% RSLogix 500 project LVD210603_BaseOnly.RSS, saved by version 12.00.00.00 %
PROJECT "LINL0619"    % processor: MicroLogix 1400 %

PROGRAM FILES
  LAD 2 "MAIN"  62 rungs  % Main Program Routine %
  LAD 4 "ENABLES"  16 rungs
  LAD 5 "FEED"  11 rungs  % normal %
  LAD 6 "SPEEDS"  11 rungs
  LAD 7 "HSC BOT"  5 rungs
  LAD 8 "HSC TOP"  5 rungs
  LAD 9 "1 MS STI"  22 rungs  % high speed %
  LAD 10 "SHIFT BOT"  5 rungs
  LAD 11 "SHIFT TOP"  6 rungs
  LAD 12 "BOTOPTIC"  3 rungs
  LAD 13 "BOTOPTMES"  7 rungs
  LAD 81 "I1"  21 rungs
  LAD 82 "I1 RESULT"  8 rungs
  LAD 83 "I1 PASS"  6 rungs
  LAD 84 "I1 FAIL"  4 rungs
  LAD 85 "I1 ACQ"  9 rungs
  LAD 86 "I1 TESTER"  5 rungs
  LAD 87 "I1 TRIG"  5 rungs
  LAD 88 "NO FIFO"  1 rungs
  LAD 89 "NO FIFO"  1 rungs
  LAD 90 "I1 DATA"  3 rungs
  LAD 91 "I1 FAULT"  9 rungs
  LAD 92 "I1 FIX1"  5 rungs
  LAD 93 "I1 FIX2"  3 rungs
  LAD 94 "I2"  1 rungs
  LAD 95 "I2 RESULT"  1 rungs
  LAD 96 "I2 PASS"  1 rungs
  LAD 97 "I2 FAIL"  1 rungs
  LAD 98 "I2 ACQ"  1 rungs
  LAD 99 "I2 TESTER"  1 rungs
  LAD 100 "I2 TRIG"  1 rungs
  LAD 101 "I2 FIFOSET"  1 rungs
  LAD 102 "I2 FIFOGET"  1 rungs
  LAD 103 "I2 DATA"  1 rungs
  LAD 104 "I2 FAULT"  1 rungs
  LAD 105 "I2 FIX1"  1 rungs
  LAD 106 "I2 FIX2"  1 rungs
  LAD 107 "I3"  1 rungs
  LAD 108 "I3 RESULT"  1 rungs
  LAD 109 "I3 PASS"  1 rungs
  LAD 110 "I3 FAIL"  1 rungs
  LAD 111 "I3 ACQ"  1 rungs
  LAD 112 "I3 TESTER"  1 rungs
  LAD 113 "I3 TRIG"  1 rungs
  LAD 114 "I3 FIFOSET"  1 rungs
  LAD 115 "I3 FIFOGET"  1 rungs
  LAD 116 "I3 DATA"  1 rungs
  LAD 117 "I3 FAULT"  1 rungs
  LAD 118 "I3 FIX1"  1 rungs
  LAD 119 "I3 FIX2"  1 rungs
  LAD 120 "I4"  1 rungs
  LAD 121 "I4 RESULT"  1 rungs
  LAD 122 "I4 PASS"  1 rungs
  LAD 123 "I4 FAIL"  1 rungs
  LAD 124 "I4 ACQ"  1 rungs
  LAD 125 "I4 TESTER"  1 rungs
  LAD 126 "I4 TRIG"  1 rungs
  LAD 127 "I4 FIFOSET"  1 rungs
  LAD 128 "I4 FIFOGET"  1 rungs
  LAD 129 "I4 DATA"  1 rungs
  LAD 130 "I4 FAULT"  1 rungs
  LAD 131 "I4 FIX1"  1 rungs
  LAD 132 "I4 FIX2"  1 rungs
  LAD 135 "XFER"  3 rungs
  LAD 137 "TOPOPTIC"  15 rungs
  LAD 138 "TOPOPVERT"  13 rungs
  LAD 139 "TOPOPREAL"  19 rungs
  LAD 140 "TOPOPTEST"  8 rungs
  LAD 141 "TOPOPRANGE"  6 rungs
  LAD 142 "TOPOPRANGE"  6 rungs
  LAD 143 "TOPOPOKAY"  6 rungs
  LAD 144 "TESTINJECT"  8 rungs
  LAD 148 "I5"  21 rungs
  LAD 149 "I5 RESULT"  7 rungs
  LAD 150 "I5 PASS"  6 rungs
  LAD 151 "I5 FAIL"  4 rungs
  LAD 152 "I5 ACQ"  9 rungs
  LAD 153 "I5 TESTER"  5 rungs
  LAD 154 "I5 TRIG"  5 rungs
  LAD 155 "I5 FIFOSET"  10 rungs
  LAD 156 "I5 FIFOGET"  8 rungs
  LAD 157 "I5 DATA"  3 rungs
  LAD 158 "I5 FAULT"  9 rungs
  LAD 159 "I5 FIX1"  5 rungs
  LAD 160 "I5 FIX2"  3 rungs
  LAD 161 "I6"  21 rungs
  LAD 162 "I6 RESULT"  7 rungs
  LAD 163 "I6 PASS"  5 rungs
  LAD 164 "I6 FAIL"  3 rungs
  LAD 165 "I6 ACQ"  8 rungs
  LAD 166 "I6 TESTER"  5 rungs
  LAD 167 "I6 TRIG"  5 rungs
  LAD 168 "I6 FIFOSET"  9 rungs
  LAD 169 "I6 FIFOGET"  8 rungs
  LAD 170 "I6 DATA"  3 rungs
  LAD 171 "I6 FAULT"  9 rungs
  LAD 172 "I6 FIX1"  5 rungs
  LAD 173 "I6 FIX2"  3 rungs
  LAD 174 "I7"  21 rungs
  LAD 175 "I7 RESULT"  7 rungs
  LAD 176 "I7 PASS"  6 rungs
  LAD 177 "I7 FAIL"  4 rungs
  LAD 178 "I7 ACQ"  9 rungs
  LAD 179 "I7 TESTER"  5 rungs
  LAD 180 "I7 TRIG"  5 rungs
  LAD 181 "I7 FIFOSET"  9 rungs
  LAD 182 "I7 FIFOGET"  8 rungs
  LAD 183 "I7 DATA"  3 rungs
  LAD 184 "I7 FAULT"  9 rungs
  LAD 185 "I7 FIX1"  5 rungs
  LAD 186 "I7 FIX2"  3 rungs
  LAD 187 "I8"  22 rungs
  LAD 188 "I8 RESULT"  7 rungs
  LAD 189 "I8 PASS"  6 rungs
  LAD 190 "I8 FAIL"  4 rungs
  LAD 191 "I8 ACQ"  9 rungs
  LAD 192 "I8 TESTER"  5 rungs
  LAD 193 "I8 TRIG"  5 rungs
  LAD 194 "I8 FIFOSET"  9 rungs
  LAD 195 "I8 FIFOGET"  8 rungs
  LAD 196 "I8 DATA"  3 rungs
  LAD 197 "I8 FAULT"  9 rungs
  LAD 198 "I8 FIX1"  5 rungs
  LAD 199 "I8 FIX2"  3 rungs
  LAD 200 "PASS BLOW"  15 rungs
  LAD 235 "TESTTRIGS"  7 rungs  % highspeed test triggers, not necessary %
  LAD 236 "TESTTRIG1"  4 rungs
  LAD 237 "TESTTRIG2"  4 rungs
  LAD 238 "TESTTRIG3"  4 rungs
  LAD 239 "TESTTRIG4"  4 rungs
  LAD 240 "TESTTRIG5"  4 rungs
  LAD 241 "TESTTRIG6"  4 rungs
  LAD 242 "TESTTRIG7"  4 rungs
  LAD 243 "TESTTRIG8"  4 rungs
  LAD 244 "PACKAGER"  31 rungs  % normal %
  LAD 245 "NO PACKAGE"  8 rungs
  LAD 246 "RATE1"  9 rungs
  LAD 247 "RATE2"  6 rungs
  LAD 248 "RESET RATE"  6 rungs
  LAD 249 "NP STOP"  8 rungs  % stop on no good %
  LAD 250 "SPEED BOT"  8 rungs  % high speed %
  LAD 251 "SPEED TOP"  8 rungs  % high speed %
  LAD 252 "P BOT"  7 rungs  % high speed %
  LAD 253 "P TOP"  7 rungs  % high speed %
  LAD 254 "TOTALCOUNT"  4 rungs
  LAD 255 "SAVED"  4 rungs

DATA FILES
  O0 OUTPUT  6 elements
  I1 INPUT  8 elements
  S2 STATUS  66 elements
  B3 BINARY  256 elements
  T4 TIMER  45 elements
  C5 COUNTER  1 elements
  R6 CONTROL  30 elements
  N7 INTEGER  200 elements
  F8 FLOAT  1 elements
  L13 LONG  256 elements
  L19 RATE DATA  50 elements
  L20 I7TIMEFIFO  50 elements
  L21 I7POSFIFO  50 elements
  L22 I8TIMEFIFO  50 elements
  L23 I8POSFIFO  50 elements
  L30 INS5TIME  50 elements
  L31 INS5POS  50 elements
  L32 INS6TIME  50 elements
  L33 INS6POS  50 elements
  B34 BOT NG  128 elements
  B35 TOP NG  128 elements
  B36 BOTGOOD  128 elements
  B37 TOPGOOD1  128 elements
  B38 EX1 TEST  128 elements
  B39 TOPGOOD2  128 elements
  B40 EX2 TEST  128 elements
  B99 REMOVED IO  5 elements
  B100 NEW HMI B  100 elements
  N101 NEW HMI N  256 elements
  L102 NEW HMI L  256 elements

LADDER 2 "MAIN"    % Main Program Routine %
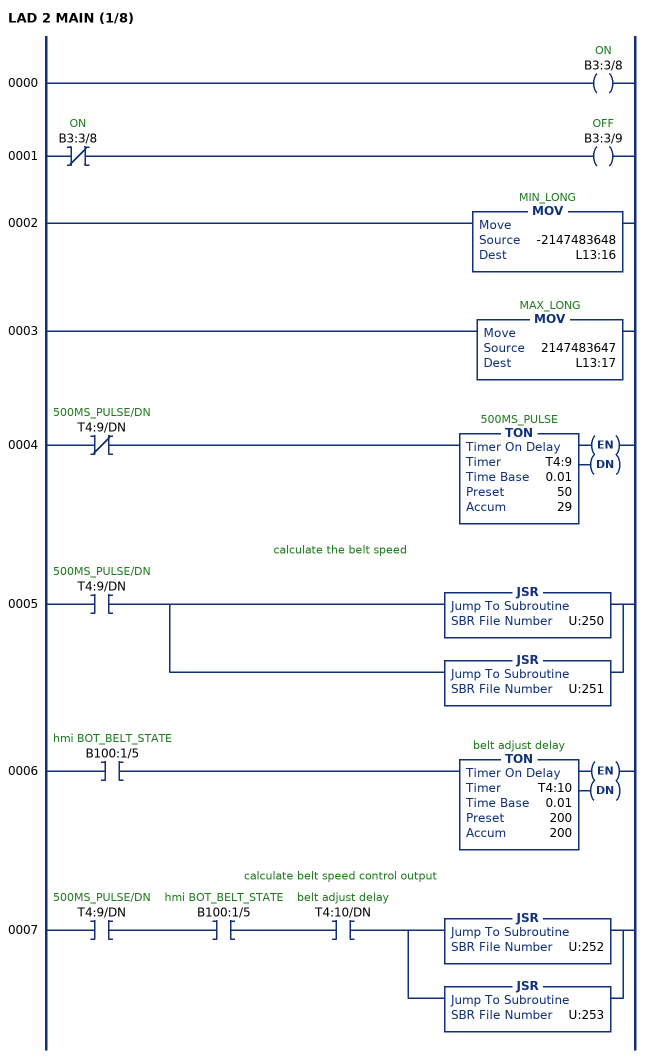
% Rung: 0 %
SOR OTE B3:3/8 EOR
%   B3:3/8  ON %
% Rung: 1 %
SOR XIO B3:3/8 OTE B3:3/9 EOR
%   B3:3/8  ON %
%   B3:3/9  OFF %
% Rung: 2 %
SOR MOV -2147483648 L13:16 EOR
%   L13:16  MIN_LONG %
% Rung: 3 %
SOR MOV 2147483647 L13:17 EOR
%   L13:17  MAX_LONG %
% Rung: 4 %
SOR XIO T4:9/DN TON T4:9 0.01 50 29 EOR
%   T4:9  500MS_PULSE %
% Rung: 5 %
% calculate the belt speed %
SOR XIC T4:9/DN BST JSR U:250 NXB JSR U:251 BND EOR
%   T4:9  500MS_PULSE %
% Rung: 6 %
SOR XIC B100:1/5 TON T4:10 0.01 200 200 EOR
%   B100:1/5  BOT_BELT_STATE  "hmi" %
%   T4:10  "belt adjust delay" %
% Rung: 7 %
% calculate belt speed control output %
SOR XIC T4:9/DN XIC B100:1/5 XIC T4:10/DN BST JSR U:252 NXB JSR U:253 BND EOR
%   T4:9  500MS_PULSE %
%   B100:1/5  BOT_BELT_STATE  "hmi" %
%   T4:10  "belt adjust delay" %

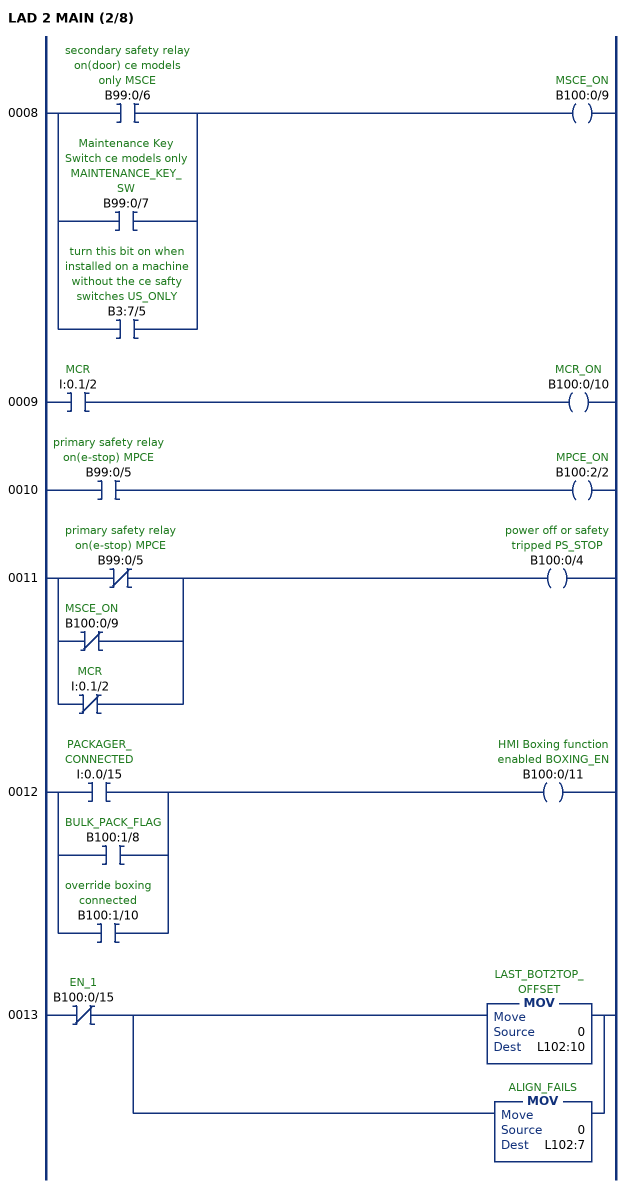
% Rung: 8 %
SOR BST XIC B99:0/6 NXB XIC B99:0/7 NXB XIC B3:7/5 BND OTE B100:0/9 EOR
%   B99:0/6  MSCE  "secondary safety relay on(door) ce models only" %
%   B99:0/7  MAINTENANCE_KEY_SW  "Maintenance Key Switch ce models only" %
%   B3:7/5  US_ONLY  "turn this bit on when installed on a machine without the ce safty switches" %
%   B100:0/9  MSCE_ON %
% Rung: 9 %
SOR XIC I:0.1/2 OTE B100:0/10 EOR
%   I:0.1/2  MCR %
%   B100:0/10  MCR_ON %
% Rung: 10 %
SOR XIC B99:0/5 OTE B100:2/2 EOR
%   B99:0/5  MPCE  "primary safety relay on(e-stop)" %
%   B100:2/2  MPCE_ON %
% Rung: 11 %
SOR BST XIO B99:0/5 NXB XIO B100:0/9 NXB XIO I:0.1/2 BND OTE B100:0/4 EOR
%   B99:0/5  MPCE  "primary safety relay on(e-stop)" %
%   B100:0/9  MSCE_ON %
%   I:0.1/2  MCR %
%   B100:0/4  PS_STOP  "power off or safety tripped" %
% Rung: 12 %
SOR BST XIC I:0.0/15 NXB XIC B100:1/8 NXB XIC B100:1/10 BND OTE B100:0/11 EOR
%   I:0.0/15  PACKAGER_CONNECTED %
%   B100:1/8  BULK_PACK_FLAG %
%   B100:1/10  "override boxing connected" %
%   B100:0/11  BOXING_EN  "HMI Boxing function enabled" %
% Rung: 13 %
SOR XIO B100:0/15 BST MOV 0 L102:10 NXB MOV 0 L102:7 BND EOR
%   B100:0/15  EN_1 %
%   L102:10  LAST_BOT2TOP_OFFSET %
%   L102:7  ALIGN_FAILS %

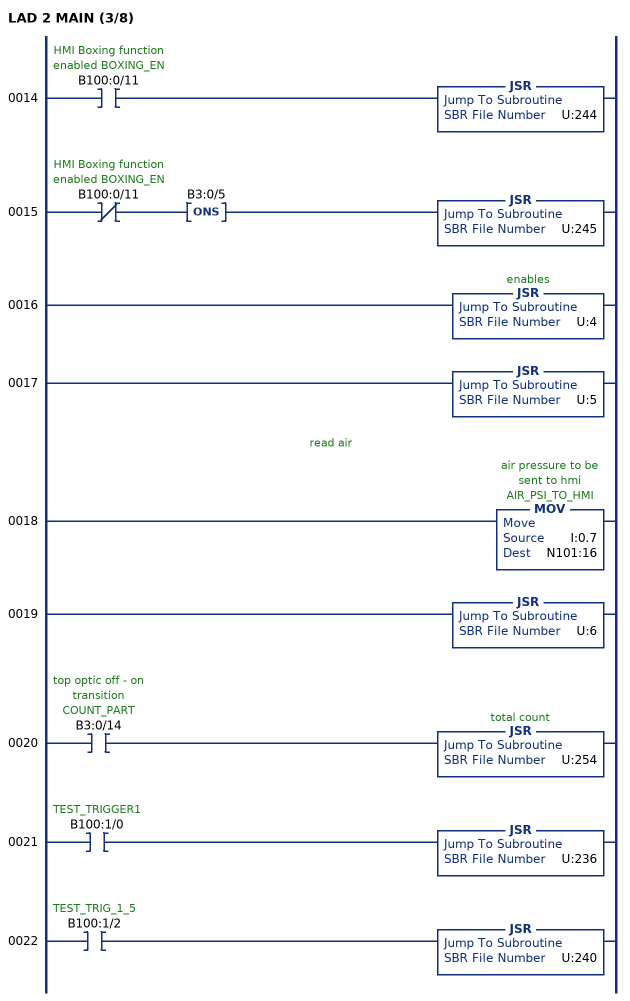
% Rung: 14 %
SOR XIC B100:0/11 JSR U:244 EOR
%   B100:0/11  BOXING_EN  "HMI Boxing function enabled" %
% Rung: 15 %
SOR XIO B100:0/11 ONS B3:0/5 JSR U:245 EOR
%   B100:0/11  BOXING_EN  "HMI Boxing function enabled" %
% Rung: 16 %
SOR JSR U:4 EOR
%   U:4  "enables" %
% Rung: 17 %
SOR JSR U:5 EOR
% Rung: 18 %
% read air %
SOR MOV I:0.7 N101:16 EOR
%   I:0.7  "Air Presure Sensor Input Signal" %
%   N101:16  AIR_PSI_TO_HMI  "air pressure to be sent to hmi" %
% Rung: 19 %
SOR JSR U:6 EOR
% Rung: 20 %
SOR XIC B3:0/14 JSR U:254 EOR
%   B3:0/14  COUNT_PART  "top optic off - on transition" %
%   U:254  "total count" %
% Rung: 21 %
SOR XIC B100:1/0 JSR U:236 EOR
%   B100:1/0  TEST_TRIGGER1 %
% Rung: 22 %
SOR XIC B100:1/2 JSR U:240 EOR
%   B100:1/2  TEST_TRIG_1_5 %

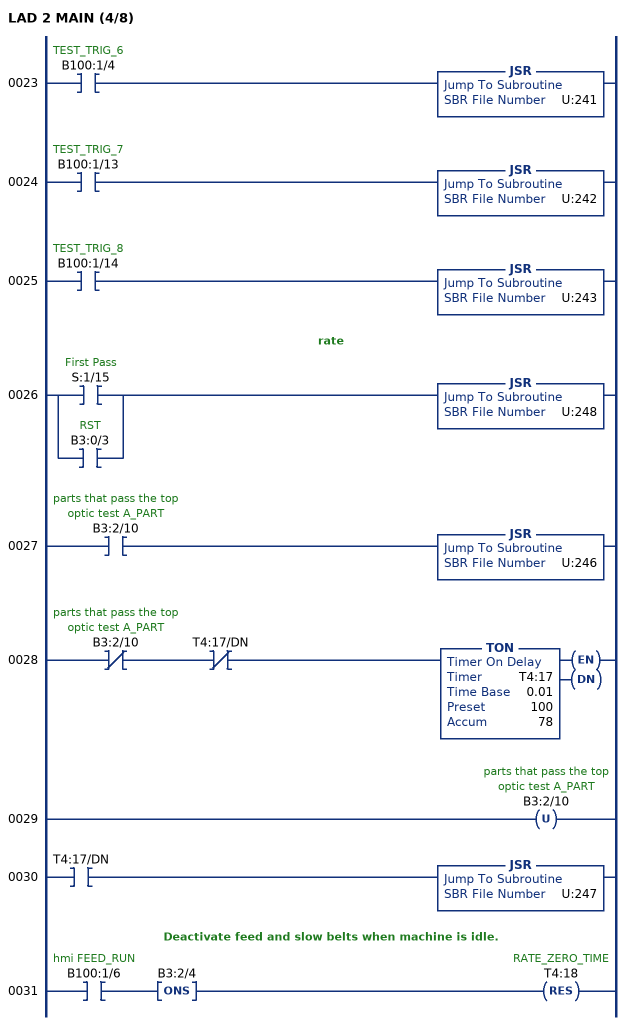
% Rung: 23 %
SOR XIC B100:1/4 JSR U:241 EOR
%   B100:1/4  TEST_TRIG_6 %
% Rung: 24 %
SOR XIC B100:1/13 JSR U:242 EOR
%   B100:1/13  TEST_TRIG_7 %
% Rung: 25 %
SOR XIC B100:1/14 JSR U:243 EOR
%   B100:1/14  TEST_TRIG_8 %
% Rung: 26 %
% TITLE: rate %
SOR BST XIC S:1/15 NXB XIC B3:0/3 BND JSR U:248 EOR
%   S:1/15  "First Pass" %
%   B3:0/3  RST %
% Rung: 27 %
SOR XIC B3:2/10 JSR U:246 EOR
%   B3:2/10  A_PART  "parts that pass the top optic test" %
% Rung: 28 %
SOR XIO B3:2/10 XIO T4:17/DN TON T4:17 0.01 100 78 EOR
%   B3:2/10  A_PART  "parts that pass the top optic test" %
% Rung: 29 %
SOR OTU B3:2/10 EOR
%   B3:2/10  A_PART  "parts that pass the top optic test" %
% Rung: 30 %
SOR XIC T4:17/DN JSR U:247 EOR
% Rung: 31 %
% TITLE: Deactivate feed and slow belts when machine is idle. %
SOR XIC B100:1/6 ONS B3:2/4 RES T4:18 EOR
%   B100:1/6  FEED_RUN  "hmi" %
%   T4:18  RATE_ZERO_TIME %

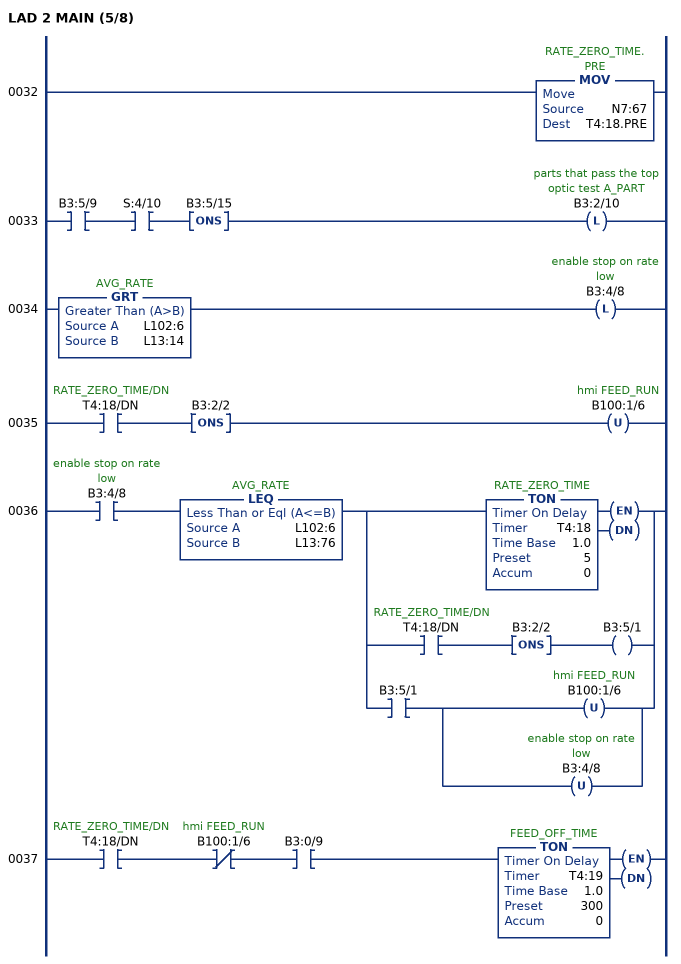
% Rung: 32 %
SOR MOV N7:67 T4:18.PRE EOR
%   N7:67  "empty bowl or jam bowl run time" %
%   T4:18  RATE_ZERO_TIME %
% Rung: 33 %
SOR XIC B3:5/9 XIC S:4/10 ONS B3:5/15 OTL B3:2/10 EOR
%   B3:2/10  A_PART  "parts that pass the top optic test" %
% Rung: 34 %
SOR GRT L102:6 L13:14 OTL B3:4/8 EOR
%   L102:6  AVG_RATE %
%   B3:4/8  "enable stop on rate low" %
% Rung: 35 %
SOR XIC T4:18/DN ONS B3:2/2 OTU B100:1/6 EOR
%   T4:18  RATE_ZERO_TIME %
%   B100:1/6  FEED_RUN  "hmi" %
% Rung: 36 %
SOR XIC B3:4/8 LEQ L102:6 L13:76 BST TON T4:18 1.0 5 0 NXB XIC T4:18/DN ONS B3:2/2 OTE B3:5/1 NXB XIC B3:5/1 BST OTU B100:1/6 NXB OTU B3:4/8 BND BND EOR
%   B3:4/8  "enable stop on rate low" %
%   L102:6  AVG_RATE %
%   T4:18  RATE_ZERO_TIME %
%   B100:1/6  FEED_RUN  "hmi" %
% Rung: 37 %
SOR XIC T4:18/DN XIO B100:1/6 XIC B3:0/9 TON T4:19 1.0 300 0 EOR
%   T4:18  RATE_ZERO_TIME %
%   B100:1/6  FEED_RUN  "hmi" %
%   T4:19  FEED_OFF_TIME %

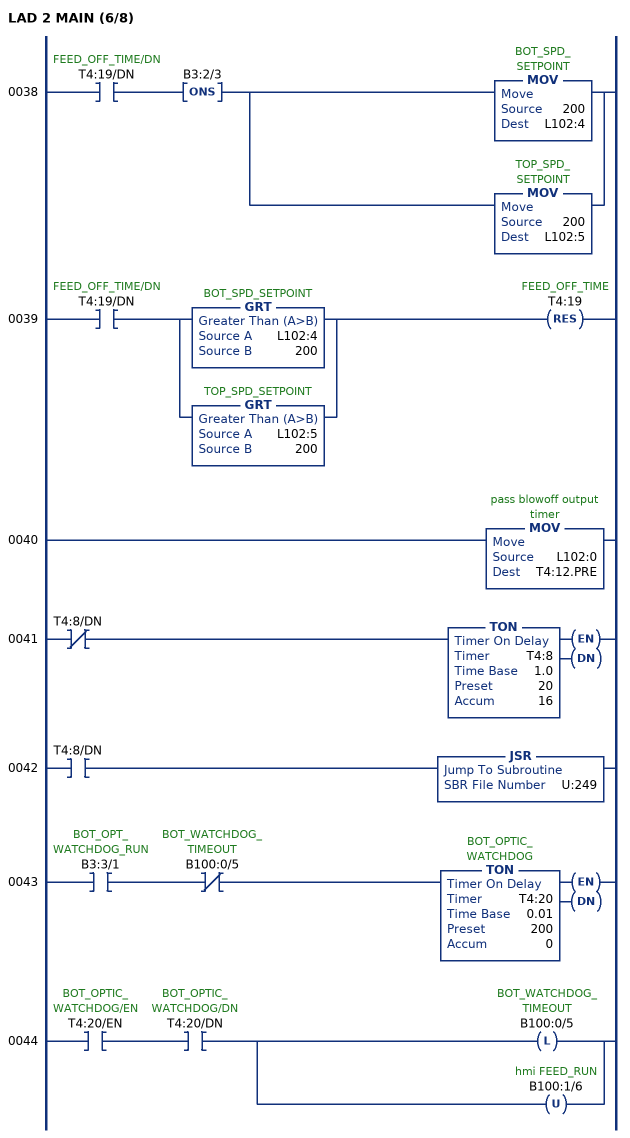
% Rung: 38 %
SOR XIC T4:19/DN ONS B3:2/3 BST MOV 200 L102:4 NXB MOV 200 L102:5 BND EOR
%   T4:19  FEED_OFF_TIME %
%   L102:4  BOT_SPD_SETPOINT %
%   L102:5  TOP_SPD_SETPOINT %
% Rung: 39 %
SOR XIC T4:19/DN BST GRT L102:4 200 NXB GRT L102:5 200 BND RES T4:19 EOR
%   T4:19  FEED_OFF_TIME %
%   L102:4  BOT_SPD_SETPOINT %
%   L102:5  TOP_SPD_SETPOINT %
% Rung: 40 %
SOR MOV L102:0 T4:12.PRE EOR
%   L102:0  BLOW_TIME %
%   T4:12  "pass blowoff output timer" %
% Rung: 41 %
SOR XIO T4:8/DN TON T4:8 1.0 20 16 EOR
% Rung: 42 %
SOR XIC T4:8/DN JSR U:249 EOR
% Rung: 43 %
SOR XIC B3:3/1 XIO B100:0/5 TON T4:20 0.01 200 0 EOR
%   B3:3/1  BOT_OPT_WATCHDOG_RUN %
%   B100:0/5  BOT_WATCHDOG_TIMEOUT %
%   T4:20  BOT_OPTIC_WATCHDOG %
% Rung: 44 %
SOR XIC T4:20/EN XIC T4:20/DN BST OTL B100:0/5 NXB OTU B100:1/6 BND EOR
%   T4:20  BOT_OPTIC_WATCHDOG %
%   B100:0/5  BOT_WATCHDOG_TIMEOUT %
%   B100:1/6  FEED_RUN  "hmi" %

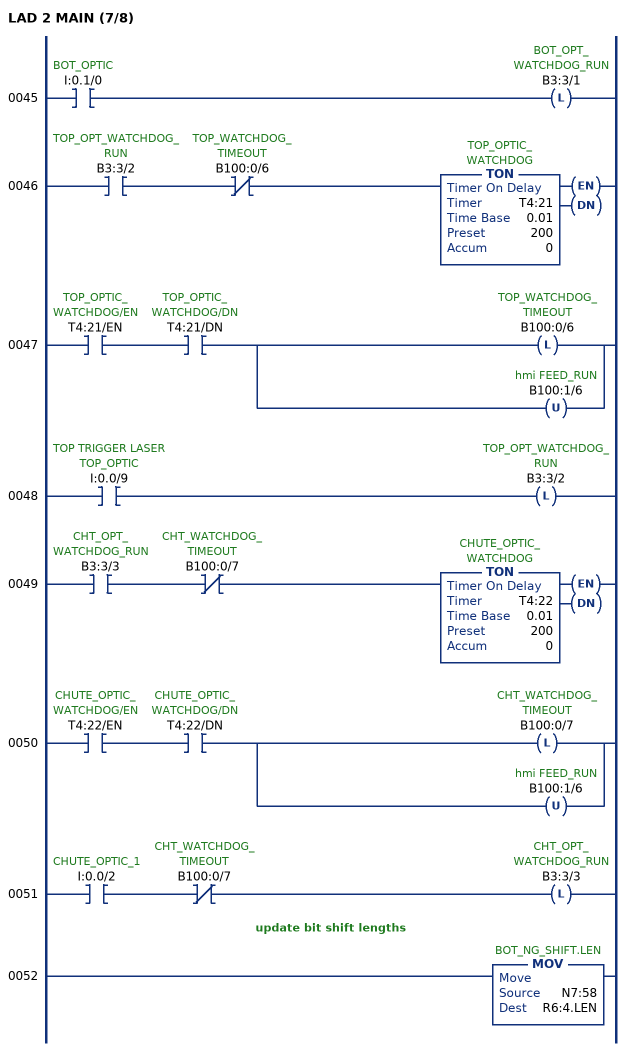
% Rung: 45 %
SOR XIC I:0.1/0 OTL B3:3/1 EOR
%   I:0.1/0  BOT_OPTIC %
%   B3:3/1  BOT_OPT_WATCHDOG_RUN %
% Rung: 46 %
SOR XIC B3:3/2 XIO B100:0/6 TON T4:21 0.01 200 0 EOR
%   B3:3/2  TOP_OPT_WATCHDOG_RUN %
%   B100:0/6  TOP_WATCHDOG_TIMEOUT %
%   T4:21  TOP_OPTIC_WATCHDOG %
% Rung: 47 %
SOR XIC T4:21/EN XIC T4:21/DN BST OTL B100:0/6 NXB OTU B100:1/6 BND EOR
%   T4:21  TOP_OPTIC_WATCHDOG %
%   B100:0/6  TOP_WATCHDOG_TIMEOUT %
%   B100:1/6  FEED_RUN  "hmi" %
% Rung: 48 %
SOR XIC I:0.0/9 OTL B3:3/2 EOR
%   I:0.0/9  TOP_OPTIC  "TOP TRIGGER LASER" %
%   B3:3/2  TOP_OPT_WATCHDOG_RUN %
% Rung: 49 %
SOR XIC B3:3/3 XIO B100:0/7 TON T4:22 0.01 200 0 EOR
%   B3:3/3  CHT_OPT_WATCHDOG_RUN %
%   B100:0/7  CHT_WATCHDOG_TIMEOUT %
%   T4:22  CHUTE_OPTIC_WATCHDOG %
% Rung: 50 %
SOR XIC T4:22/EN XIC T4:22/DN BST OTL B100:0/7 NXB OTU B100:1/6 BND EOR
%   T4:22  CHUTE_OPTIC_WATCHDOG %
%   B100:0/7  CHT_WATCHDOG_TIMEOUT %
%   B100:1/6  FEED_RUN  "hmi" %
% Rung: 51 %
SOR XIC I:0.0/2 XIO B100:0/7 OTL B3:3/3 EOR
%   I:0.0/2  CHUTE_OPTIC_1 %
%   B100:0/7  CHT_WATCHDOG_TIMEOUT %
%   B3:3/3  CHT_OPT_WATCHDOG_RUN %
% Rung: 52 %
% TITLE: update bit shift lengths %
SOR MOV N7:58 R6:4.LEN EOR
%   N7:58  BOT_NG_LENGTH %
%   R6:4  BOT_NG_SHIFT %

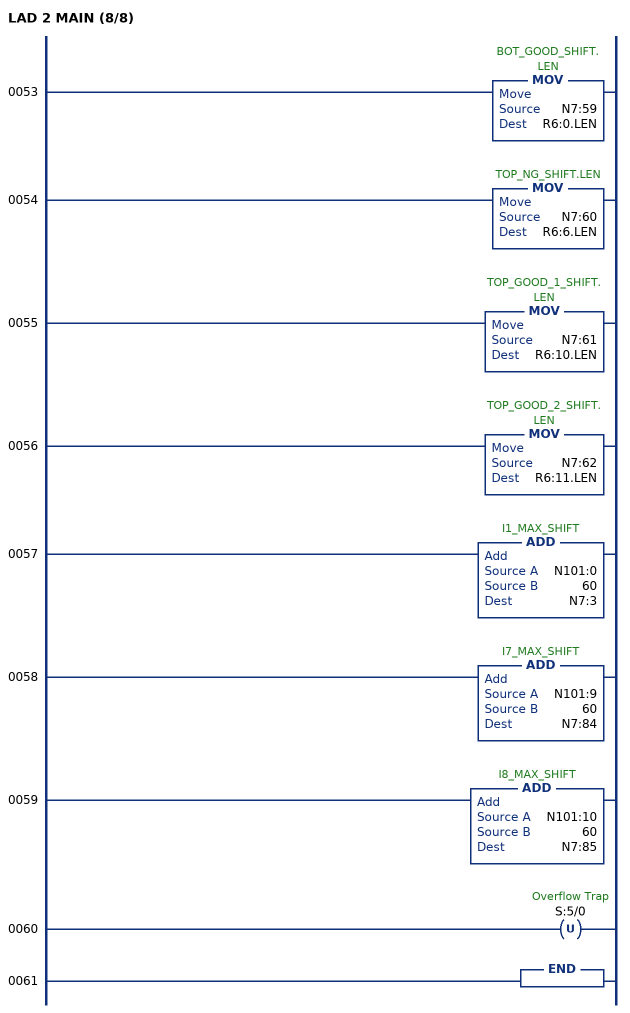
% Rung: 53 %
SOR MOV N7:59 R6:0.LEN EOR
%   N7:59  BOT_GOOD_LENGTH %
%   R6:0  BOT_GOOD_SHIFT %
% Rung: 54 %
SOR MOV N7:60 R6:6.LEN EOR
%   N7:60  TOP_NG_LENGTH %
%   R6:6  TOP_NG_SHIFT %
% Rung: 55 %
SOR MOV N7:61 R6:10.LEN EOR
%   N7:61  TOP_GOOD1_LENGTH %
%   R6:10  TOP_GOOD_1_SHIFT %
% Rung: 56 %
SOR MOV N7:62 R6:11.LEN EOR
%   N7:62  TOP_GOOD2_LENGTH %
%   R6:11  TOP_GOOD_2_SHIFT %
% Rung: 57 %
SOR ADD N101:0 60 N7:3 EOR
%   N101:0  I1_TRIG_LOC %
%   N7:3  I1_MAX_SHIFT %
% Rung: 58 %
SOR ADD N101:9 60 N7:84 EOR
%   N101:9  I7_TRIG_LOC %
%   N7:84  I7_MAX_SHIFT %
% Rung: 59 %
SOR ADD N101:10 60 N7:85 EOR
%   N101:10  I8_TRIG_LOC %
%   N7:85  I8_MAX_SHIFT %
% Rung: 60 %
SOR OTU S:5/0 EOR
%   S:5/0  "Overflow Trap" %
% Rung: 61 %
SOR END EOR

LADDER 4 "ENABLES"
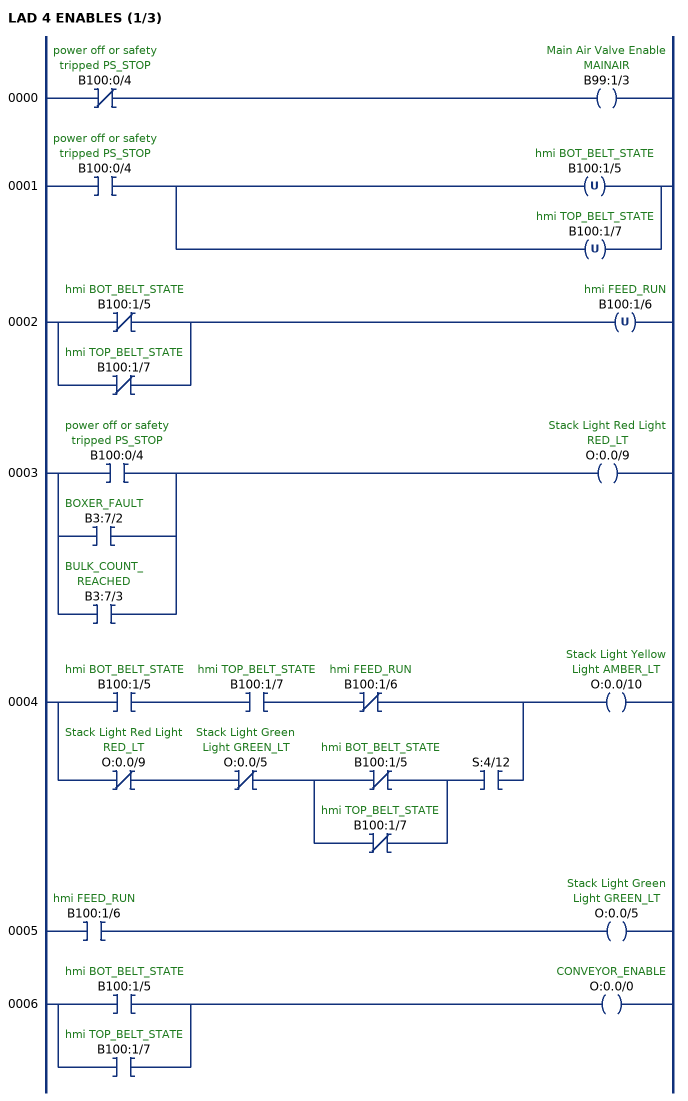
% Rung: 0 %
SOR XIO B100:0/4 OTE B99:1/3 EOR
%   B100:0/4  PS_STOP  "power off or safety tripped" %
%   B99:1/3  MAINAIR  "Main Air Valve Enable" %
% Rung: 1 %
SOR XIC B100:0/4 BST OTU B100:1/5 NXB OTU B100:1/7 BND EOR
%   B100:0/4  PS_STOP  "power off or safety tripped" %
%   B100:1/5  BOT_BELT_STATE  "hmi" %
%   B100:1/7  TOP_BELT_STATE  "hmi" %
% Rung: 2 %
SOR BST XIO B100:1/5 NXB XIO B100:1/7 BND OTU B100:1/6 EOR
%   B100:1/5  BOT_BELT_STATE  "hmi" %
%   B100:1/7  TOP_BELT_STATE  "hmi" %
%   B100:1/6  FEED_RUN  "hmi" %
% Rung: 3 %
SOR BST XIC B100:0/4 NXB XIC B3:7/2 NXB XIC B3:7/3 BND OTE O:0.0/9 EOR
%   B100:0/4  PS_STOP  "power off or safety tripped" %
%   B3:7/2  BOXER_FAULT %
%   B3:7/3  BULK_COUNT_REACHED %
%   O:0.0/9  RED_LT  "Stack Light Red Light" %
% Rung: 4 %
SOR BST XIC B100:1/5 XIC B100:1/7 XIO B100:1/6 NXB XIO O:0.0/9 XIO O:0.0/5 BST XIO B100:1/5 NXB XIO B100:1/7 BND XIC S:4/12 BND OTE O:0.0/10 EOR
%   B100:1/5  BOT_BELT_STATE  "hmi" %
%   B100:1/7  TOP_BELT_STATE  "hmi" %
%   B100:1/6  FEED_RUN  "hmi" %
%   O:0.0/9  RED_LT  "Stack Light Red Light" %
%   O:0.0/5  GREEN_LT  "Stack Light Green Light" %
%   O:0.0/10  AMBER_LT  "Stack Light Yellow Light" %
% Rung: 5 %
SOR XIC B100:1/6 OTE O:0.0/5 EOR
%   B100:1/6  FEED_RUN  "hmi" %
%   O:0.0/5  GREEN_LT  "Stack Light Green Light" %
% Rung: 6 %
SOR BST XIC B100:1/5 NXB XIC B100:1/7 BND OTE O:0.0/0 EOR
%   B100:1/5  BOT_BELT_STATE  "hmi" %
%   B100:1/7  TOP_BELT_STATE  "hmi" %
%   O:0.0/0  CONVEYOR_ENABLE %

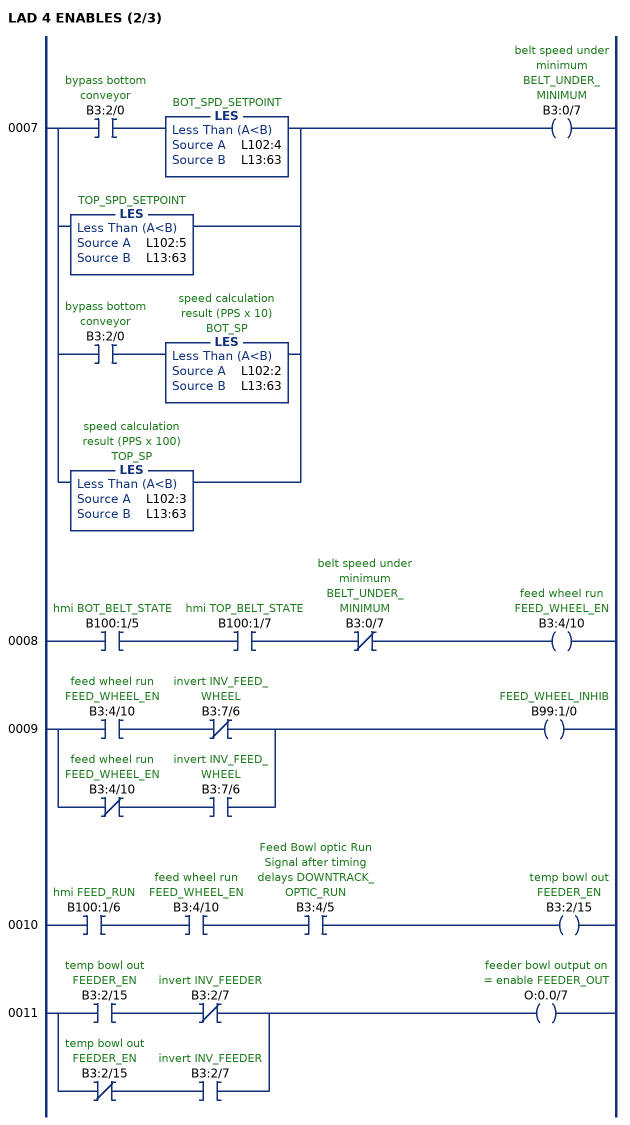
% Rung: 7 %
SOR BST XIC B3:2/0 LES L102:4 L13:63 NXB LES L102:5 L13:63 NXB XIC B3:2/0 LES L102:2 L13:63 NXB LES L102:3 L13:63 BND OTE B3:0/7 EOR
%   B3:2/0  "bypass bottom conveyor" %
%   L102:4  BOT_SPD_SETPOINT %
%   L13:63  "min belt speed" %
%   L102:5  TOP_SPD_SETPOINT %
%   L102:2  BOT_SP  "speed calculation result (PPS x 10)" %
%   L102:3  TOP_SP  "speed calculation result (PPS x 100)" %
%   B3:0/7  BELT_UNDER_MINIMUM  "belt speed under minimum" %
% Rung: 8 %
SOR XIC B100:1/5 XIC B100:1/7 XIO B3:0/7 OTE B3:4/10 EOR
%   B100:1/5  BOT_BELT_STATE  "hmi" %
%   B100:1/7  TOP_BELT_STATE  "hmi" %
%   B3:0/7  BELT_UNDER_MINIMUM  "belt speed under minimum" %
%   B3:4/10  FEED_WHEEL_EN  "feed wheel run" %
% Rung: 9 %
SOR BST XIC B3:4/10 XIO B3:7/6 NXB XIO B3:4/10 XIC B3:7/6 BND OTE B99:1/0 EOR
%   B3:4/10  FEED_WHEEL_EN  "feed wheel run" %
%   B3:7/6  INV_FEED_WHEEL  "invert" %
%   B99:1/0  FEED_WHEEL_INHIB %
% Rung: 10 %
SOR XIC B100:1/6 XIC B3:4/10 XIC B3:4/5 OTE B3:2/15 EOR
%   B100:1/6  FEED_RUN  "hmi" %
%   B3:4/10  FEED_WHEEL_EN  "feed wheel run" %
%   B3:4/5  DOWNTRACK_OPTIC_RUN  "Feed Bowl optic Run Signal after timing delays" %
%   B3:2/15  FEEDER_EN  "temp bowl out" %
% Rung: 11 %
SOR BST XIC B3:2/15 XIO B3:2/7 NXB XIO B3:2/15 XIC B3:2/7 BND OTE O:0.0/7 EOR
%   B3:2/15  FEEDER_EN  "temp bowl out" %
%   B3:2/7  INV_FEEDER  "invert" %
%   O:0.0/7  FEEDER_OUT  "feeder bowl output on = enable" %

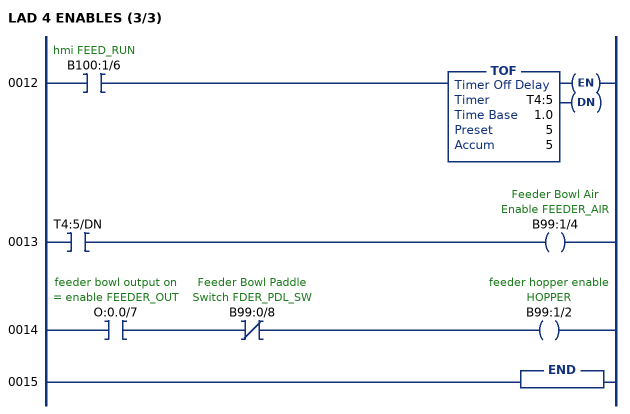
% Rung: 12 %
SOR XIC B100:1/6 TOF T4:5 1.0 5 5 EOR
%   B100:1/6  FEED_RUN  "hmi" %
% Rung: 13 %
SOR XIC T4:5/DN OTE B99:1/4 EOR
%   B99:1/4  FEEDER_AIR  "Feeder Bowl Air Enable" %
% Rung: 14 %
SOR XIC O:0.0/7 XIO B99:0/8 OTE B99:1/2 EOR
%   O:0.0/7  FEEDER_OUT  "feeder bowl output on = enable" %
%   B99:0/8  FDER_PDL_SW  "Feeder Bowl Paddle Switch" %
%   B99:1/2  HOPPER  "feeder hopper enable" %
% Rung: 15 %
SOR END EOR

LADDER 5 "FEED"    % normal %
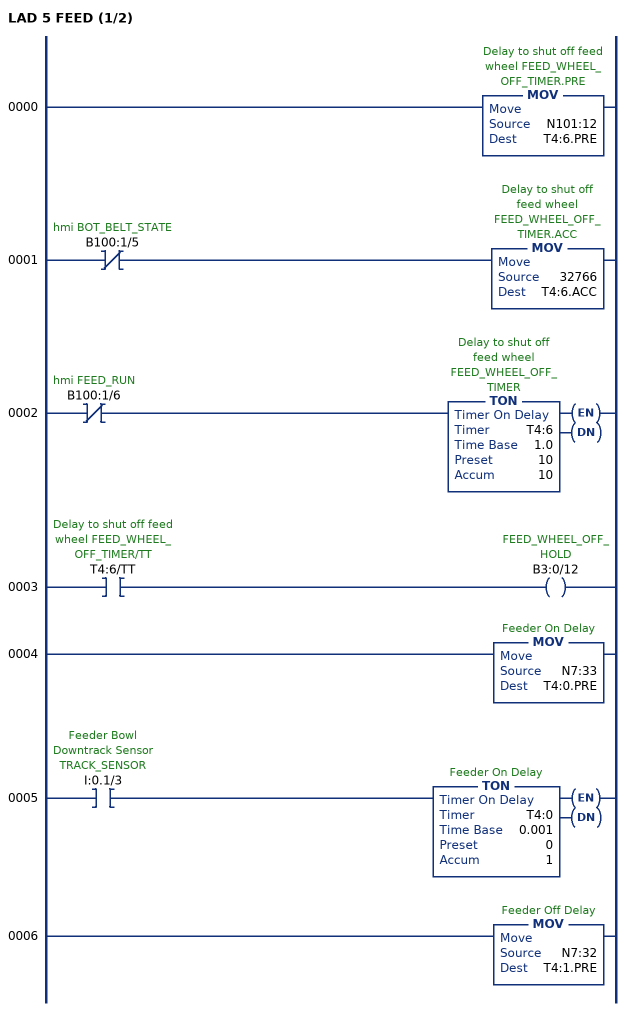
% Rung: 0 %
SOR MOV N101:12 T4:6.PRE EOR
%   N101:12  FEED_WHEEL_STOP_TIME %
%   T4:6  FEED_WHEEL_OFF_TIMER  "Delay to shut off feed wheel" %
% Rung: 1 %
SOR XIO B100:1/5 MOV 32766 T4:6.ACC EOR
%   B100:1/5  BOT_BELT_STATE  "hmi" %
%   T4:6  FEED_WHEEL_OFF_TIMER  "Delay to shut off feed wheel" %
% Rung: 2 %
SOR XIO B100:1/6 TON T4:6 1.0 10 10 EOR
%   B100:1/6  FEED_RUN  "hmi" %
%   T4:6  FEED_WHEEL_OFF_TIMER  "Delay to shut off feed wheel" %
% Rung: 3 %
SOR XIC T4:6/TT OTE B3:0/12 EOR
%   T4:6  FEED_WHEEL_OFF_TIMER  "Delay to shut off feed wheel" %
%   B3:0/12  FEED_WHEEL_OFF_HOLD %
% Rung: 4 %
SOR MOV N7:33 T4:0.PRE EOR
%   N7:33  "down track on delay" %
%   T4:0  "Feeder On Delay" %
% Rung: 5 %
SOR XIC I:0.1/3 TON T4:0 0.001 0 1 EOR
%   I:0.1/3  TRACK_SENSOR  "Feeder Bowl Downtrack Sensor" %
%   T4:0  "Feeder On Delay" %
% Rung: 6 %
SOR MOV N7:32 T4:1.PRE EOR
%   N7:32  "down track off delay" %
%   T4:1  "Feeder Off Delay" %

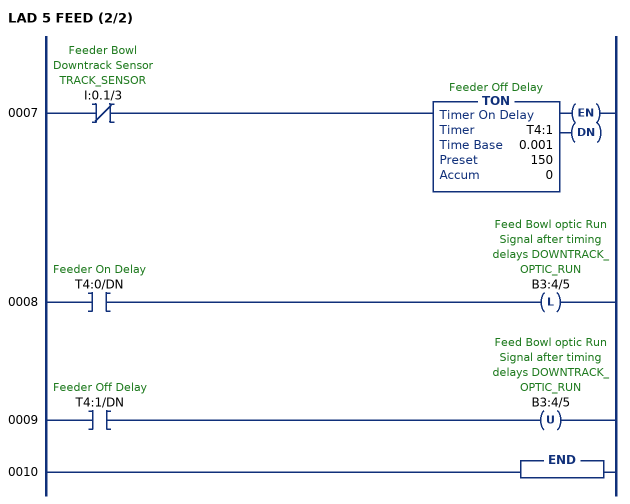
% Rung: 7 %
SOR XIO I:0.1/3 TON T4:1 0.001 150 0 EOR
%   I:0.1/3  TRACK_SENSOR  "Feeder Bowl Downtrack Sensor" %
%   T4:1  "Feeder Off Delay" %
% Rung: 8 %
SOR XIC T4:0/DN OTL B3:4/5 EOR
%   T4:0  "Feeder On Delay" %
%   B3:4/5  DOWNTRACK_OPTIC_RUN  "Feed Bowl optic Run Signal after timing delays" %
% Rung: 9 %
SOR XIC T4:1/DN OTU B3:4/5 EOR
%   T4:1  "Feeder Off Delay" %
%   B3:4/5  DOWNTRACK_OPTIC_RUN  "Feed Bowl optic Run Signal after timing delays" %
% Rung: 10 %
SOR END EOR

LADDER 6 "SPEEDS"
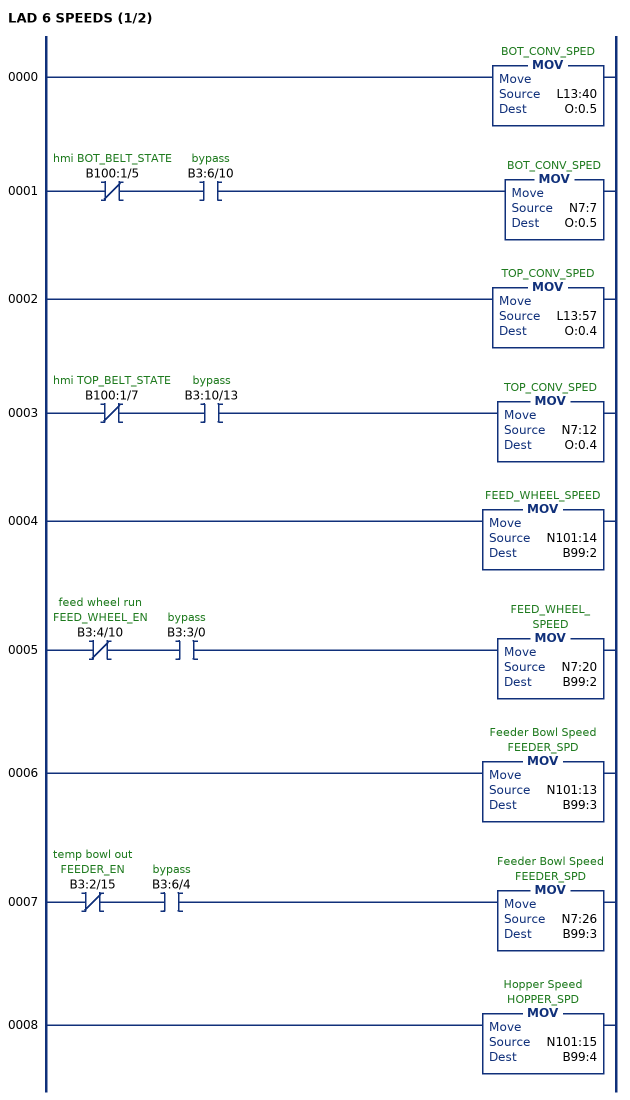
% Rung: 0 %
SOR MOV L13:40 O:0.5 EOR
%   L13:40  SCALED_BOT_VALUE %
%   O:0.5  BOT_CONV_SPED %
% Rung: 1 %
SOR XIO B100:1/5 XIC B3:6/10 MOV N7:7 O:0.5 EOR
%   B100:1/5  BOT_BELT_STATE  "hmi" %
%   B3:6/10  "bypass" %
%   O:0.5  BOT_CONV_SPED %
% Rung: 2 %
SOR MOV L13:57 O:0.4 EOR
%   L13:57  SCALED_TOP_VALUE %
%   O:0.4  TOP_CONV_SPED %
% Rung: 3 %
SOR XIO B100:1/7 XIC B3:10/13 MOV N7:12 O:0.4 EOR
%   B100:1/7  TOP_BELT_STATE  "hmi" %
%   B3:10/13  "bypass" %
%   O:0.4  TOP_CONV_SPED %
% Rung: 4 %
SOR MOV N101:14 B99:2 EOR
%   N101:14  FEED_WHL_SPD_SET  "feed wheel speed setting from hmi" %
%   B99:2  FEED_WHEEL_SPEED %
% Rung: 5 %
SOR XIO B3:4/10 XIC B3:3/0 MOV N7:20 B99:2 EOR
%   B3:4/10  FEED_WHEEL_EN  "feed wheel run" %
%   B3:3/0  "bypass" %
%   B99:2  FEED_WHEEL_SPEED %
% Rung: 6 %
SOR MOV N101:13 B99:3 EOR
%   N101:13  FEED_BOWL_SET_SPD %
%   B99:3  FEEDER_SPD  "Feeder Bowl Speed" %
% Rung: 7 %
SOR XIO B3:2/15 XIC B3:6/4 MOV N7:26 B99:3 EOR
%   B3:2/15  FEEDER_EN  "temp bowl out" %
%   B3:6/4  "bypass" %
%   B99:3  FEEDER_SPD  "Feeder Bowl Speed" %
% Rung: 8 %
SOR MOV N101:15 B99:4 EOR
%   N101:15  HOPPER_SPD_SET  "hopper speed setting from hmi" %
%   B99:4  HOPPER_SPD  "Hopper Speed" %

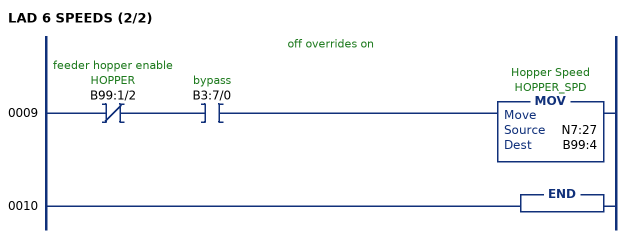
% Rung: 9 %
% off overrides on %
SOR XIO B99:1/2 XIC B3:7/0 MOV N7:27 B99:4 EOR
%   B99:1/2  HOPPER  "feeder hopper enable" %
%   B3:7/0  "bypass" %
%   B99:4  HOPPER_SPD  "Hopper Speed" %
% Rung: 10 %
SOR END EOR

LADDER 7 "HSC BOT"
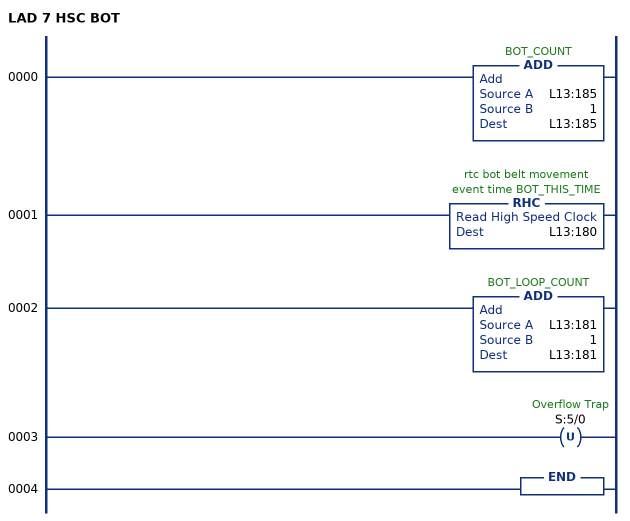
% Rung: 0 %
SOR ADD L13:185 1 L13:185 EOR
%   L13:185  BOT_COUNT %
% Rung: 1 %
SOR RHC L13:180 EOR
%   L13:180  BOT_THIS_TIME  "rtc bot belt movement event time" %
% Rung: 2 %
SOR ADD L13:181 1 L13:181 EOR
%   L13:181  BOT_LOOP_COUNT %
% Rung: 3 %
SOR OTU S:5/0 EOR
%   S:5/0  "Overflow Trap" %
% Rung: 4 %
SOR END EOR

LADDER 8 "HSC TOP"
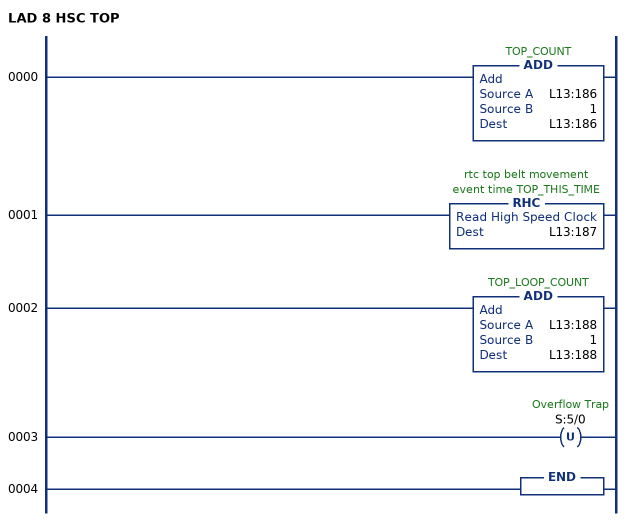
% Rung: 0 %
SOR ADD L13:186 1 L13:186 EOR
%   L13:186  TOP_COUNT %
% Rung: 1 %
SOR RHC L13:187 EOR
%   L13:187  TOP_THIS_TIME  "rtc top belt movement event time" %
% Rung: 2 %
SOR ADD L13:188 1 L13:188 EOR
%   L13:188  TOP_LOOP_COUNT %
% Rung: 3 %
SOR OTU S:5/0 EOR
%   S:5/0  "Overflow Trap" %
% Rung: 4 %
SOR END EOR

LADDER 9 "1 MS STI"    % high speed %
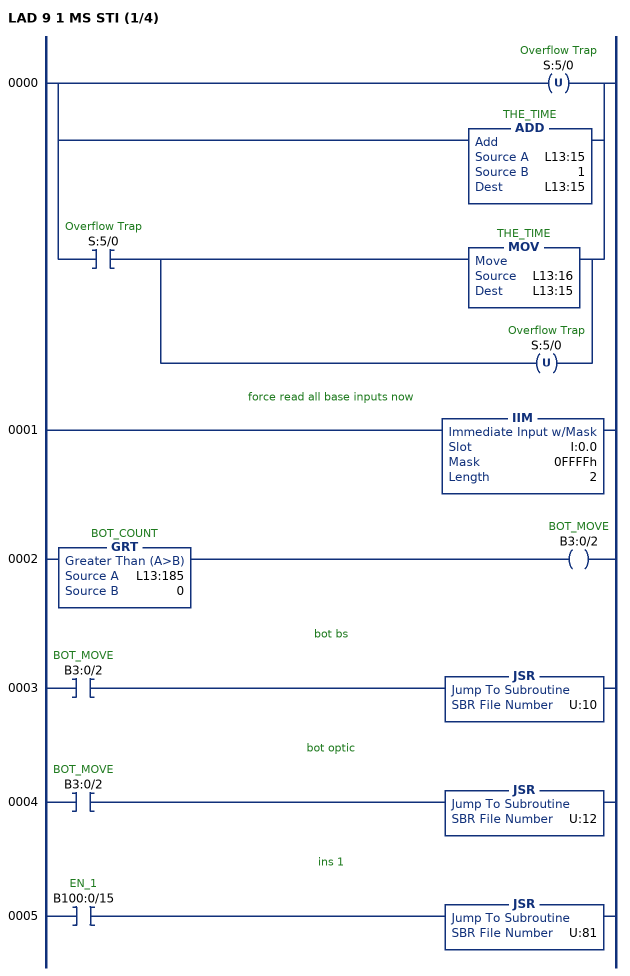
% Rung: 0 %
SOR BST OTU S:5/0 NXB ADD L13:15 1 L13:15 NXB XIC S:5/0 BST MOV L13:16 L13:15 NXB OTU S:5/0 BND BND EOR
%   S:5/0  "Overflow Trap" %
%   L13:15  THE_TIME %
%   L13:16  MIN_LONG %
% Rung: 1 %
% force read all base inputs now %
SOR IIM I:0.0 0FFFFh 2 EOR
% Rung: 2 %
SOR GRT L13:185 0 OTE B3:0/2 EOR
%   L13:185  BOT_COUNT %
%   B3:0/2  BOT_MOVE %
% Rung: 3 %
% bot bs %
SOR XIC B3:0/2 JSR U:10 EOR
%   B3:0/2  BOT_MOVE %
% Rung: 4 %
% bot optic %
SOR XIC B3:0/2 JSR U:12 EOR
%   B3:0/2  BOT_MOVE %
% Rung: 5 %
% ins 1 %
SOR XIC B100:0/15 JSR U:81 EOR
%   B100:0/15  EN_1 %

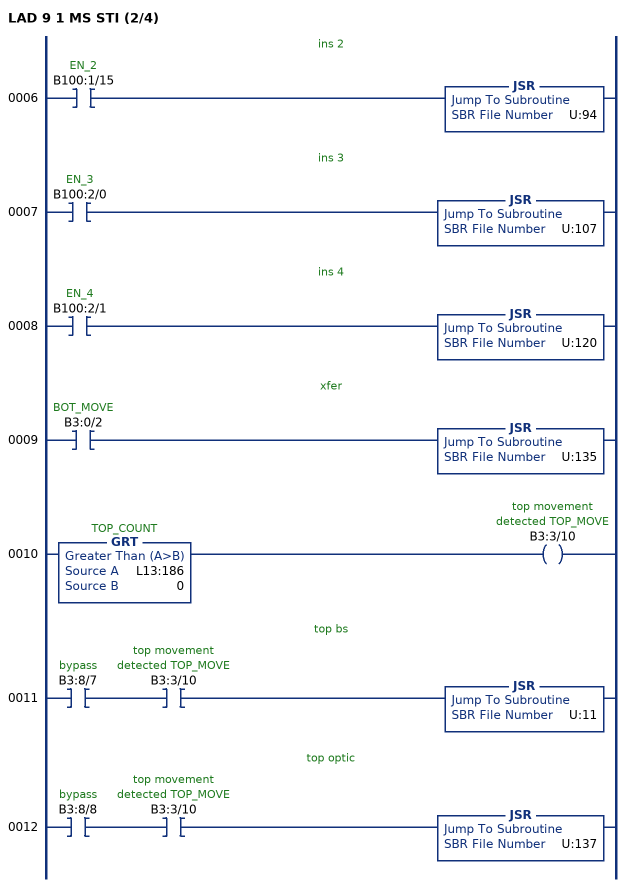
% Rung: 6 %
% ins 2 %
SOR XIC B100:1/15 JSR U:94 EOR
%   B100:1/15  EN_2 %
% Rung: 7 %
% ins 3 %
SOR XIC B100:2/0 JSR U:107 EOR
%   B100:2/0  EN_3 %
% Rung: 8 %
% ins 4 %
SOR XIC B100:2/1 JSR U:120 EOR
%   B100:2/1  EN_4 %
% Rung: 9 %
% xfer %
SOR XIC B3:0/2 JSR U:135 EOR
%   B3:0/2  BOT_MOVE %
% Rung: 10 %
SOR GRT L13:186 0 OTE B3:3/10 EOR
%   L13:186  TOP_COUNT %
%   B3:3/10  TOP_MOVE  "top movement detected" %
% Rung: 11 %
% top bs %
SOR XIC B3:8/7 XIC B3:3/10 JSR U:11 EOR
%   B3:8/7  "bypass" %
%   B3:3/10  TOP_MOVE  "top movement detected" %
% Rung: 12 %
% top optic %
SOR XIC B3:8/8 XIC B3:3/10 JSR U:137 EOR
%   B3:8/8  "bypass" %
%   B3:3/10  TOP_MOVE  "top movement detected" %

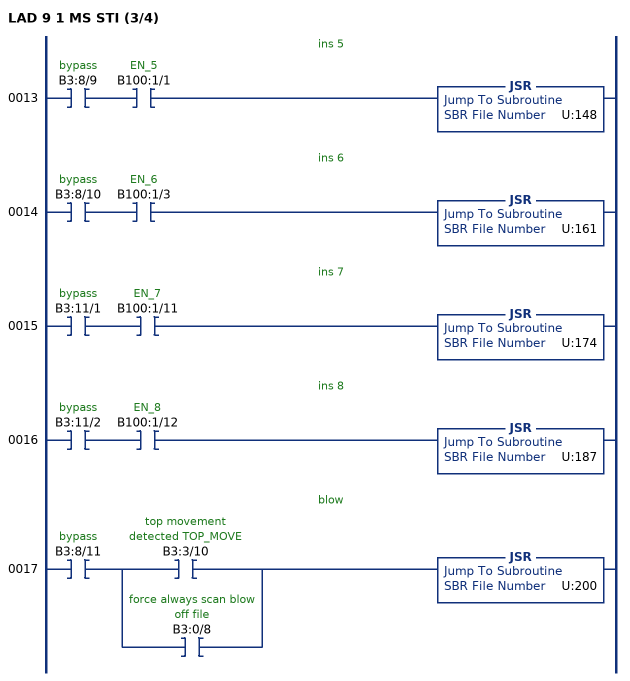
% Rung: 13 %
% ins 5 %
SOR XIC B3:8/9 XIC B100:1/1 JSR U:148 EOR
%   B3:8/9  "bypass" %
%   B100:1/1  EN_5 %
% Rung: 14 %
% ins 6 %
SOR XIC B3:8/10 XIC B100:1/3 JSR U:161 EOR
%   B3:8/10  "bypass" %
%   B100:1/3  EN_6 %
% Rung: 15 %
% ins 7 %
SOR XIC B3:11/1 XIC B100:1/11 JSR U:174 EOR
%   B3:11/1  "bypass" %
%   B100:1/11  EN_7 %
% Rung: 16 %
% ins 8 %
SOR XIC B3:11/2 XIC B100:1/12 JSR U:187 EOR
%   B3:11/2  "bypass" %
%   B100:1/12  EN_8 %
% Rung: 17 %
% blow %
SOR XIC B3:8/11 BST XIC B3:3/10 NXB XIC B3:0/8 BND JSR U:200 EOR
%   B3:8/11  "bypass" %
%   B3:3/10  TOP_MOVE  "top movement detected" %
%   B3:0/8  "force always scan blow off file" %

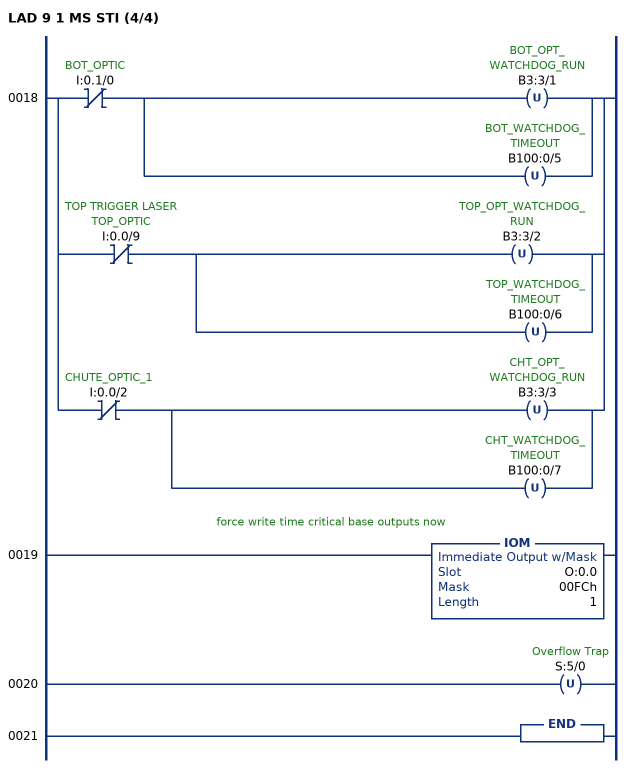
% Rung: 18 %
SOR BST XIO I:0.1/0 BST OTU B3:3/1 NXB OTU B100:0/5 BND NXB XIO I:0.0/9 BST OTU B3:3/2 NXB OTU B100:0/6 BND NXB XIO I:0.0/2 BST OTU B3:3/3 NXB OTU B100:0/7 BND BND EOR
%   I:0.1/0  BOT_OPTIC %
%   B3:3/1  BOT_OPT_WATCHDOG_RUN %
%   B100:0/5  BOT_WATCHDOG_TIMEOUT %
%   I:0.0/9  TOP_OPTIC  "TOP TRIGGER LASER" %
%   B3:3/2  TOP_OPT_WATCHDOG_RUN %
%   B100:0/6  TOP_WATCHDOG_TIMEOUT %
%   I:0.0/2  CHUTE_OPTIC_1 %
%   B3:3/3  CHT_OPT_WATCHDOG_RUN %
%   B100:0/7  CHT_WATCHDOG_TIMEOUT %
% Rung: 19 %
% force write time critical base outputs now %
SOR IOM O:0.0 00FCh 1 EOR
% Rung: 20 %
SOR OTU S:5/0 EOR
%   S:5/0  "Overflow Trap" %
% Rung: 21 %
SOR END EOR

LADDER 10 "SHIFT BOT"
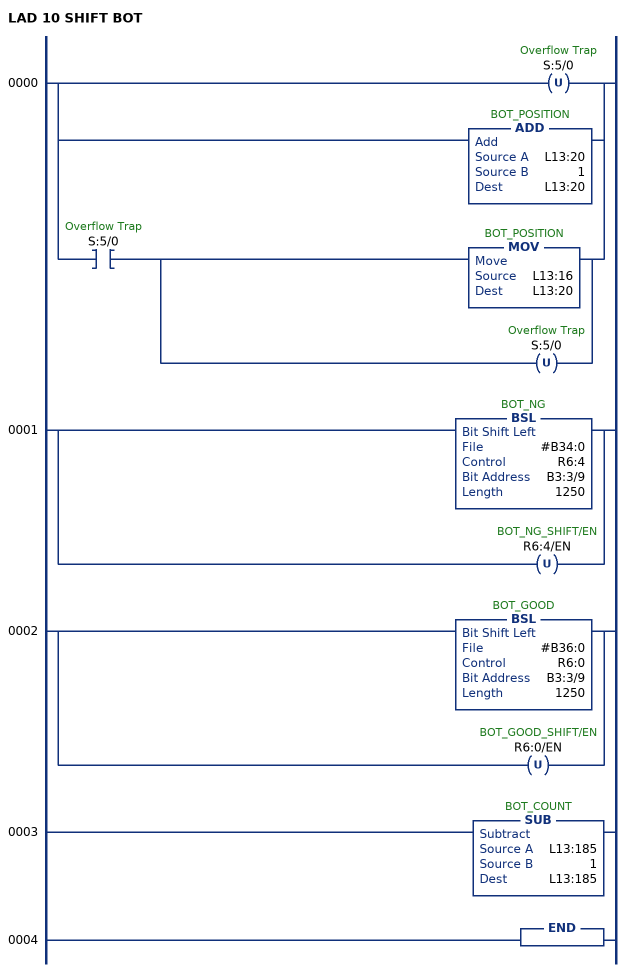
% Rung: 0 %
SOR BST OTU S:5/0 NXB ADD L13:20 1 L13:20 NXB XIC S:5/0 BST MOV L13:16 L13:20 NXB OTU S:5/0 BND BND EOR
%   S:5/0  "Overflow Trap" %
%   L13:20  BOT_POSITION %
%   L13:16  MIN_LONG %
% Rung: 1 %
SOR BST BSL #B34:0 R6:4 B3:3/9 1250 NXB OTU R6:4/EN BND EOR
%   B34:0  BOT_NG %
%   R6:4  BOT_NG_SHIFT %
%   B3:3/9  OFF %
% Rung: 2 %
SOR BST BSL #B36:0 R6:0 B3:3/9 1250 NXB OTU R6:0/EN BND EOR
%   B36:0  BOT_GOOD %
%   R6:0  BOT_GOOD_SHIFT %
%   B3:3/9  OFF %
% Rung: 3 %
SOR SUB L13:185 1 L13:185 EOR
%   L13:185  BOT_COUNT %
% Rung: 4 %
SOR END EOR

LADDER 11 "SHIFT TOP"
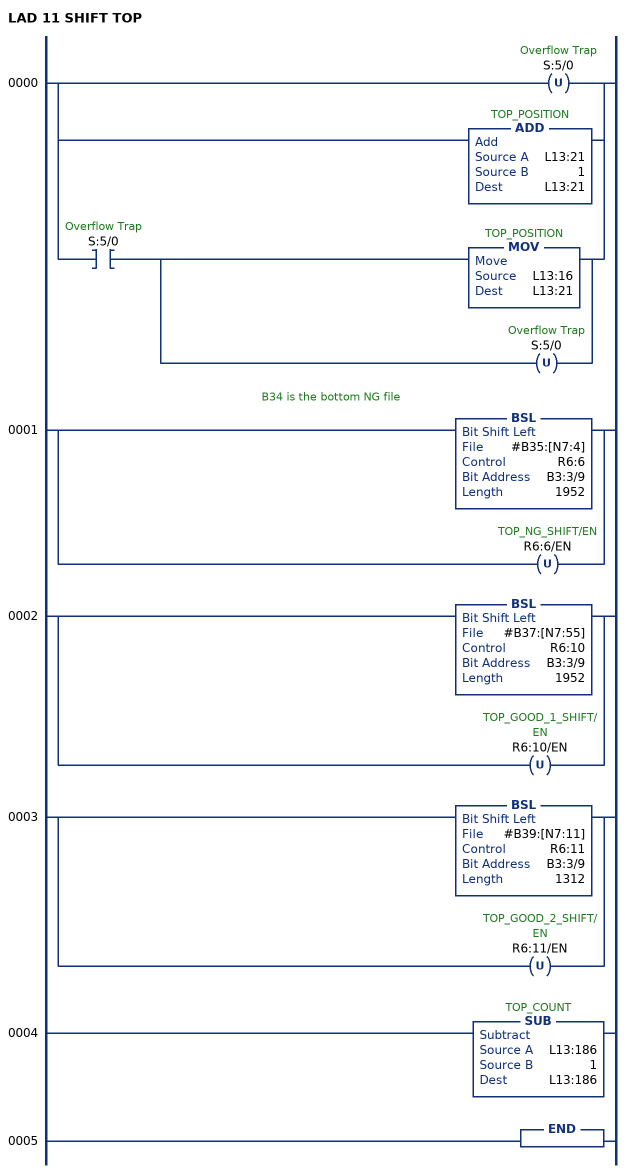
% Rung: 0 %
SOR BST OTU S:5/0 NXB ADD L13:21 1 L13:21 NXB XIC S:5/0 BST MOV L13:16 L13:21 NXB OTU S:5/0 BND BND EOR
%   S:5/0  "Overflow Trap" %
%   L13:21  TOP_POSITION %
%   L13:16  MIN_LONG %
% Rung: 1 %
% B34 is the bottom NG file %
SOR BST BSL #B35:[N7:4] R6:6 B3:3/9 1952 NXB OTU R6:6/EN BND EOR
%   N7:4  TOP_NG_START_WORD %
%   R6:6  TOP_NG_SHIFT %
%   B3:3/9  OFF %
% Rung: 2 %
SOR BST BSL #B37:[N7:55] R6:10 B3:3/9 1952 NXB OTU R6:10/EN BND EOR
%   N7:55  TOP_GOOD1_START_WORD %
%   R6:10  TOP_GOOD_1_SHIFT %
%   B3:3/9  OFF %
% Rung: 3 %
SOR BST BSL #B39:[N7:11] R6:11 B3:3/9 1312 NXB OTU R6:11/EN BND EOR
%   N7:11  TOP_GOOD2_START_WORD %
%   R6:11  TOP_GOOD_2_SHIFT %
%   B3:3/9  OFF %
% Rung: 4 %
SOR SUB L13:186 1 L13:186 EOR
%   L13:186  TOP_COUNT %
% Rung: 5 %
SOR END EOR

LADDER 12 "BOTOPTIC"
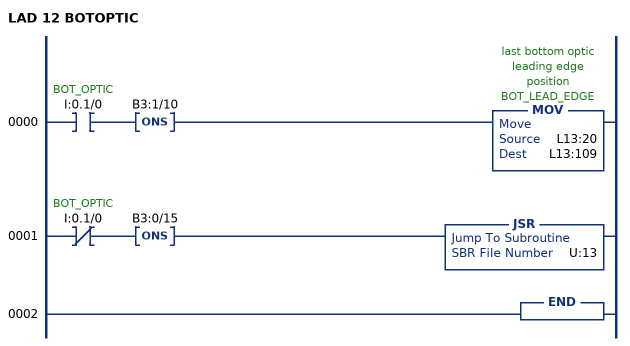
% Rung: 0 %
SOR XIC I:0.1/0 ONS B3:1/10 MOV L13:20 L13:109 EOR
%   I:0.1/0  BOT_OPTIC %
%   L13:20  BOT_POSITION %
%   L13:109  BOT_LEAD_EDGE  "last bottom optic leading edge position" %
% Rung: 1 %
SOR XIO I:0.1/0 ONS B3:0/15 JSR U:13 EOR
%   I:0.1/0  BOT_OPTIC %
% Rung: 2 %
SOR END EOR

LADDER 13 "BOTOPTMES"
